FUNCTION_BLOCK FB_HE_SATT_FindOptimalCombination
VAR
    iFilterHolder1 : I_HE_SATT_FilterHolder;
    iFilterHolder2 : I_HE_SATT_FilterHolder;
    iFilterHolder3 : I_HE_SATT_FilterHolder;
    iFilterHolder4 : I_HE_SATT_FilterHolder;
    iFilterHolder5 : I_HE_SATT_FilterHolder;
//     iCalculateSiliconThickness : I_CalculateThickness;
//     iCalculateDiamondThickness : I_CalculateThickness;
//     iCalculateGermaniumThickness : I_CalculateThickness;
END_VAR


METHOD PUBLIC FindOptimalCombination
VAR_INPUT
	(* [0.0 - 1.0]*)
	fRequestedTransmission	: LREAL;
	eRequestedRoundingMode	: E_HE_SATT_RoundingMode;
	fRequestedAllowableTolerance	: LREAL;
    iFilterCombinationCollector : I_HE_SATT_FilterCombinationCollector;
END_VAR
VAR_OUTPUT
    bWithinAllowableTolerance : BOOL;
    iOptimalCombination : I_HE_SATT_FilterCombination;
END_VAR
END_METHOD

END_FUNCTION_BLOCK

(* stored: Version 1.1.0.1
   POU FB_HE_SATT_FindOptimalCombination: Id {03a9882a-fdb5-4066-a35a-05d3adec64d5}, SpecialFunc None
   Method FindOptimalCombination: Id {11772ad2-35e1-4e17-8c00-98ae190f53b5} *)
